FUNCTION_BLOCK FB_MotionAxisNC IMPLEMENTS I_MotionAxis
VAR_INPUT
END_VAR
VAR_OUTPUT
END_VAR
VAR
    {attribute 'no_copy'}
    AxisRef : REFERENCE TO AXIS_REF;
    iMotionAxisCommon : I_MotionAxisCommon;
    iPersistentDataStorage : I_PersistentDataStorage;
    iMotionLogger : I_MotionLogger;

    stAxisParameterSetExposed : ST_AxisParameterSetExposed;

    // This prevent unexpected logical 1 on stMotionStage.bExecute
    nErrorId			: UDINT:=0;
    bHomingBusy			: BOOL;
    bHomingDone			: BOOL;
    fHomePosition : LREAL :=0.0;
    bError				: BOOL;
    sErrorMessage		: STRING;

    fSetPosition	: LREAL;
    fSetVelocity	: LREAL;
    fSetAcceleration	: LREAL := 0.0;
    fSetDeceleration	: LREAL := 0.0;
    fSetJerk	: LREAL := 0.0;
    nHomingMode:ENUM_EpicsHomeCmd :=ENUM_EpicsHomeCmd.NONE;
    eBufferMode	: MC_BufferMode := .MC_BufferMode.MC_Aborting;
    eMoveMode : E_MoveMode;
    sName : STRING;
    // Piezo Motion Control
    tholtime		: TIME := T#10S;
    bBusy : BOOL;
    bDone: BOOL;
    bPowerEnable : BOOL;
    bPowerEnableNegative : BOOL;
    bPowerEnablePositive : BOOL;
    bPowerIsEnabled : BOOL;
    fPowerOverride : LREAL;
    bResetDone : BOOL;
    bHaltDone : BOOL;
    bHomeDone  : BOOL;

    {attribute 'hide'}
    eAxisState : MC_AxisStates;
    // intermediary motion signal: from EPICS interface
    bCmdMoveAbsolute	: BOOL;
    bCmdReset 			: BOOL;
    bCmdHalt 			: BOOL;
    bCmdMoveHome			: BOOL;
    nCommand 		: UINT;
    nCommandData		: UINT;
    nEncoderCount	: UDINT;
    fMoveAbsoluteTargetPosition : LREAL;
    fMoveAbsoluteTargetVelocity : LREAL;
    fMoveAbsoluteTargetAcceleration : LREAL;
    fMoveAbsoluteTargetDeceleration : LREAL;
    fMoveAbsoluteTargetJerk : LREAL;
    fMeasuredAcceleration : LREAL;
    fMeasuredVelocity : LREAL;
    fMeasuredPosition : LREAL;
    fMeasuredPositionDiff : LREAL;

    rtDone 				: R_TRIG;
    rtError				: R_TRIG;
    rtReset				: R_TRIG;
    rtHomed				: R_TRIG;
    ftServo				: F_TRIG;
END_VAR

// Propagate user command to common worker
// 1- Power status
iMotionAxisCOmmon.BufferMode := THIS^.eBufferMode;
iMotionAxisCommon.PowerEnable := THIS^.bPowerEnable;
iMotionAxisCommon.PowerEnableNegative := THIS^.bPowerEnableNegative;
iMotionAxisCommon.PowerEnablePositive := THIS^.bPowerEnablePositive;
iMotionAxisCommon.PowerOverride := THIS^.fPowerOverride;
// 2- Motion commands
iMotionAxisCommon.CommandedHalt := THIS^.bCmdHalt;
iMotionAxisCommon.CommandedReset := THIS^.bCmdReset;
iMotionAxisCommon.CommandedMoveAbsolute := THIS^.bCmdMoveAbsolute;
iMotionAxisCommon.MoveAbsoluteTargetPosition := THIS^.fMoveAbsoluteTargetPosition;
iMotionAxisCommon.MoveAbsoluteTargetVelocity := THIS^.fMoveAbsoluteTargetVelocity;
iMotionAxisCommon.MoveAbsoluteTargetAcceleration := THIS^.fMoveAbsoluteTargetAcceleration;
iMotionAxisCommon.MoveAbsoluteTargetDeceleration := THIS^.fMoveAbsoluteTargetDeceleration;
iMotionAxisCommon.MoveAbsoluteTargetJerk := THIS^.fMoveAbsoluteTargetJerk;

// readbacks and status update from common worker
THIS^.fMeasuredAcceleration := iMotionAxisCommon.MeasuredAcceleration;
THIS^.fMeasuredVelocity := iMotionAxisCommon.MeasuredVelocity;
THIS^.fMeasuredPosition := iMotionAxisCommon.MeasuredPosition;
THIS^.fMeasuredPositionDiff := iMotionAxisCommon.MeasuredPositionDiff;
THIS^.bHaltDone := iMotionAxisCommon.HaltDone;
THIS^.bResetDone := iMotionAxisCommon.ResetDone;
THIS^.bDone := iMotionAxisCommon.MoveAbsoluteDone OR THIS^.HomeDone;
THIS^.bBusy := iMotionAxisCommon.MoveAbsoluteBusy OR THIS^.HomingBusy;
THIS^.bError := iMotionAxisCommon.Error;
THIS^.nErrorId := iMotionAxisCommon.ErrorID;
THIS^.sErrorMessage := iMotionAxisCommon.ErrorMessage;
THIS^.eAxisState := iMotionAxisCommon.AxisState;

// reset cmds if done, error or reset
rtDone(CLK:=bDone);
rtError(CLK:=bError);
rtReset(CLK:=bCmdReset);
IF rtDone.Q OR rtError.Q OR rtReset.Q THEN
    bCmdMoveAbsolute	:= FALSE;
    bCmdReset	:= FALSE;
    bCmdHalt 	:= FALSE;
    bCmdMoveHome	:= FALSE;
END_IF

PROPERTY AxisParameterSetExposed : ST_AxisParameterSetExposed
GET
AxisParameterSetExposed := stAxisParameterSetExposed;
END_GET
END_PROPERTY

PROPERTY AxisState : MC_AxisStates
GET
AxisState := eAxisState;
END_GET
END_PROPERTY

{warning 'Add property implementation'}
PROPERTY BufferMode : MC_BufferMode
SET
BufferMode := eBufferMode;
END_SET
END_PROPERTY

PROPERTY Busy : BOOL
GET
Busy := bBusy;
END_GET
END_PROPERTY

PROPERTY CmdHalt : BOOL
GET
CmdHalt := bCmdHalt;
END_GET
SET
bCmdHalt := CmdHalt;
END_SET
END_PROPERTY

PROPERTY CmdMoveAbsolute : BOOL
GET
CmdMoveAbsolute := bCmdMoveAbsolute;
END_GET
SET
bCmdMoveAbsolute := CmdMoveAbsolute;
END_SET
END_PROPERTY

PROPERTY CmdMoveHome : BOOL
GET
CmdMoveHome := bCmdMoveHome;
END_GET
SET
bCmdMoveHome := CmdMoveHome;
END_SET
END_PROPERTY


PROPERTY CmdReset : BOOL
GET
CmdReset := bCmdReset;
END_GET
SET
bCmdReset := CmdReset;
END_SET
END_PROPERTY

PROPERTY Command : UINT
SET
END_SET
END_PROPERTY

PROPERTY CommandData : UINT
SET
nCommandData := CommandData;
END_SET
END_PROPERTY

PROPERTY Done : BOOL
GET
Done := bDone;
END_GET
END_PROPERTY

PROPERTY EncoderCount : UDINT
GET
EncoderCount := nEncoderCount;
END_GET
END_PROPERTY

PROPERTY Error : BOOL
GET
Error := bError;
END_GET
END_PROPERTY

{warning 'Add property implementation'}
PROPERTY ErrorID : UDINT
GET
ErrorID := nErrorID;
END_GET
END_PROPERTY

{warning 'Add property implementation'}
PROPERTY ErrorMessage : STRING
GET
ErrorMessage := sErrorMessage;
END_GET
END_PROPERTY

//FB_Init is always available implicitly and it is used primarily for initialization.
//The return value is not evaluated. For a specific influence, you can also declare the
//methods explicitly and provide additional code there with the standard initialization
//code. You can evaluate the return value.
METHOD FB_Init: BOOL
VAR_INPUT
    bInitRetains: BOOL; // TRUE: the retain variables are initialized (reset warm / reset cold)
    bInCopyCode: BOOL;  // TRUE: the instance will be copied to the copy code afterward (online change)

    AxisRef : REFERENCE TO AXIS_REF;
    iMotionAxisCommon : I_MotionAxisCommon;
    iPersistentDataStorage : I_PersistentDataStorage;
    iMotionLogger : I_MotionLogger;
END_VAR
THIS^.AxisRef REF= AxisRef;
THIS^.iMotionAxisCommon := iMotionAxisCommon;
THIS^.iPersistentDataStorage := iPersistentDataStorage;
THIS^.iMotionLogger := iMotionLogger;
END_METHOD

PROPERTY HaltDone : BOOL
GET
HaltDone := bHaltDone;
END_GET
END_PROPERTY

{warning 'Add property implementation'}
PROPERTY HomeDone : BOOL
GET
END_GET
END_PROPERTY

{warning 'Add property implementation'}
PROPERTY HomeMode : E_EpicsHomeCmd
GET
END_GET
SET
END_SET
END_PROPERTY

{warning 'Add property implementation'}
PROPERTY HomePosition : LREAL
GET
END_GET
SET
END_SET
END_PROPERTY

{warning 'Add property implementation'}
PROPERTY HomingBusy : BOOL
GET
END_GET
SET
END_SET
END_PROPERTY

{warning 'Add method implementation '}
METHOD InterruptMove
END_METHOD

PROPERTY MeasuredAcceleration : LREAL
GET
MeasuredAcceleration := fMeasuredAcceleration;
END_GET
END_PROPERTY

{warning 'Add property implementation'}
PROPERTY MeasuredPosition : LREAL
GET
MeasuredPosition := fMeasuredPosition;
END_GET
END_PROPERTY

{warning 'Add property implementation'}
PROPERTY MeasuredPositionDiff : LREAL
GET
MeasuredPositionDiff := fMeasuredPositionDiff;
END_GET
END_PROPERTY

PROPERTY MeasuredVelocity : LREAL
GET
MeasuredVelocity := fMeasuredVelocity;
END_GET
END_PROPERTY

{warning 'Add property implementation'}
PROPERTY ModeOfOperation : SINT
GET
END_GET
SET
END_SET
END_PROPERTY

PROPERTY MoveAbsoluteTargetAcceleration : LREAL
GET
MoveAbsoluteTargetAcceleration := fMoveAbsoluteTargetAcceleration;
END_GET
SET
fMoveAbsoluteTargetAcceleration := MoveAbsoluteTargetAcceleration;
END_SET
END_PROPERTY

PROPERTY MoveAbsoluteTargetDeceleration : LREAL
GET
MoveAbsoluteTargetDeceleration := fMoveAbsoluteTargetDeceleration;
END_GET
SET
fMoveAbsoluteTargetDeceleration := MoveAbsoluteTargetDeceleration;
END_SET
END_PROPERTY

PROPERTY MoveAbsoluteTargetJerk : LREAL
GET
MoveAbsoluteTargetJerk := fMoveAbsoluteTargetJerk;
END_GET
SET
fMoveAbsoluteTargetJerk := MoveAbsoluteTargetJerk;
END_SET
END_PROPERTY

PROPERTY MoveAbsoluteTargetPosition : LREAL
GET
MoveAbsoluteTargetPosition := fMoveAbsoluteTargetPosition;
END_GET
SET
fMoveAbsoluteTargetPosition := MoveAbsoluteTargetPosition;
END_SET
END_PROPERTY

PROPERTY MoveAbsoluteTargetVelocity : LREAL
GET
MoveAbsoluteTargetVelocity := fMoveAbsoluteTargetVelocity;
END_GET
SET
fMoveAbsoluteTargetVelocity := MoveAbsoluteTargetVelocity;
END_SET
END_PROPERTY

PROPERTY MoveMode : E_MoveMode
GET
MoveMode := eMoveMode;
END_GET
SET
eMoveMode := MoveMode;
END_SET
END_PROPERTY

PROPERTY Name : STRING
GET
Name := sName;
END_GET
SET
sName := Name;
END_SET
END_PROPERTY

{warning 'Add property implementation'}
PROPERTY NegativeMotionIsEnabled : BOOL
GET
END_GET
END_PROPERTY

{warning 'Add property implementation'}
PROPERTY PositiveMotionIsEnabled : BOOL
GET
END_GET
END_PROPERTY

PROPERTY PowerEnable : BOOL
GET
PowerEnable := bPowerEnable;
END_GET
SET
bPowerEnable := PowerEnable;
END_SET
END_PROPERTY

PROPERTY PowerEnableNegative : BOOL
GET
PowerEnableNegative := bPowerEnableNegative;
END_GET
SET
bPowerEnableNegative := PowerEnableNegative;
END_SET
END_PROPERTY

PROPERTY PowerEnablePositive : BOOL
GET
PowerEnablePositive := bPowerEnablePositive;
END_GET
SET
bPowerEnablePositive := PowerEnablePositive;
END_SET
END_PROPERTY

{warning 'Add property implementation'}
PROPERTY PowerIsEnabled : BOOL
GET
PowerIsEnabled := bPowerIsEnabled;
END_GET
END_PROPERTY

{warning 'Add property implementation'}
PROPERTY PowerOverride : LREAL
GET
PowerOverride := fPowerOverride;
END_GET
SET
fPowerOverride := PowerOverride;
END_SET
END_PROPERTY

PROPERTY ResetDone : BOOL
GET
ResetDone := bResetDone ;
END_GET
END_PROPERTY

{warning 'Add property implementation'}
PROPERTY Servo : BOOL
GET
END_GET
SET
END_SET
END_PROPERTY

(*
    Check all post condition before updating bCommandedMoveAbsolute
    The implmentatation will depend on the axis type
    DS402 NC/Direct axis : Implementation need to check that the drive is in the correct mode before initaiting the move then set bCommandedMoveAbsolute
    MP NC axis : will immediately write to bCommandedMoveAbsolute
*)
METHOD StartMove : BOOL
VAR_INPUT
END_VAR
CASE eMoveMode OF
    E_MoveMode.DISCRETE:
        iMotionAxisCommon.CommandedMoveAbsolute := THIS^.bCmdMoveAbsolute;
    E_MoveMode.HOMING:
    THIS^.bCmdMoveHome := TRUE;
END_CASE

// for typical NC axis no further test is needed
StartMove := TRUE;
END_METHOD

{warning 'Add method implementation '}
METHOD StopMove
END_METHOD

END_FUNCTION_BLOCK

(* stored: Version 1.1.0.1
   POU FB_MotionAxisNC: Id {abd0b982-5130-4244-8207-eba0b3246906}, SpecialFunc None
   Property AxisParameterSetExposed: Id {384b2d0e-5f4f-4936-8350-ceae816b150e}
   Get Get: Id {c87f54a1-a5eb-49de-8441-7a2ad0ec72de}
   Property AxisState: Id {904290e4-8519-49b9-badc-b3e1713daec6}
   Get Get: Id {ccec9d39-634d-4098-ae3d-57765a8e4217}
   Property BufferMode: Id {2c65028d-a104-4e19-872f-4dd701e61531}
   Set Set: Id {6e4cbde5-d3db-4fb0-90d0-8e798f99604b}
   Property Busy: Id {8b5e8894-c876-41b1-9e2c-980090299d06}
   Get Get: Id {0589f453-0019-4df2-87e7-619c947d4d89}
   Property CmdHalt: Id {18dd0b55-37ec-4bc8-a0d2-55b6db6a152f}
   Get Get: Id {a8673054-4564-489f-91d8-dc779daec553}
   Set Set: Id {bb6fa02c-7a76-469a-ae3d-d5fddedf6fd7}
   Property CmdMoveAbsolute: Id {8ba6543e-9bbe-4c2c-985e-e7797189c137}
   Get Get: Id {10aedfd5-412b-492b-b988-266d9f40addf}
   Set Set: Id {1edbd315-9001-4619-ac2e-1d29105a5138}
   Property CmdMoveHome: Id {9dc329c6-3e63-4e47-98ec-522d097b78c3}
   Get Get: Id {497b21ae-b468-49fa-a678-10ae542a591a}
   Set Set: Id {d15709fd-f925-450c-9e97-7665b59292b5}
   Property CmdReset: Id {70bf962c-f201-42b0-acce-f42a534f0e53}
   Get Get: Id {400e310e-bcfd-485d-b2ea-e2b29fff54cb}
   Set Set: Id {d260d983-2678-4bcb-9070-7db5839a6fca}
   Property Command: Id {1bfbf561-216d-484d-b0f5-59e0d5d323f0}
   Set Set: Id {7b937c3c-33f5-4681-a1fc-8827e5918112}
   Property CommandData: Id {2f61ec8e-7923-460c-bb0d-1c4f6bf683f9}
   Set Set: Id {7ac59737-5819-446b-adb3-fad8bc24c252}
   Property Done: Id {7dfea87f-91d0-4696-931e-3f0a58f16ac5}
   Get Get: Id {b56b7cc9-86b2-4c3c-bc8f-26dc7bf2e509}
   Property EncoderCount: Id {cd5917d9-7633-485a-80ea-f12e3b700502}
   Get Get: Id {929c4496-fbe3-4004-b896-c4d0a35e2293}
   Property Error: Id {4da1c0dd-304a-4f96-9c35-e21861c7cc5a}
   Get Get: Id {cb4df7cd-44c4-45b9-9d32-a492dc206cc9}
   Property ErrorID: Id {a9cd6d81-3a12-4ea6-a064-5e3b63b03982}
   Get Get: Id {5ddc443f-6d54-4a83-a527-83e86fdb72b0}
   Property ErrorMessage: Id {aeeaa0d1-15f3-4400-b508-44a15c83d1d3}
   Get Get: Id {5f52a084-10af-4e78-8941-03dd3f8cdb45}
   Method FB_Init: Id {0f22422e-d0d7-4f19-ba6a-909d8434ca89}
   Property HaltDone: Id {3e07c920-60e0-4810-a3dc-4b8f36ba148b}
   Get Get: Id {fbe1db8b-e303-42af-aa5c-f6f6b3b3c9b9}
   Property HomeDone: Id {58d55820-86b5-4ff6-b9aa-fa09a9de7d99}
   Get Get: Id {260eedc9-efbe-40a9-af5a-fbf7edde8655}
   Property HomeMode: Id {66c6b98c-e856-4ec1-8f29-50ec1e680ce0}
   Get Get: Id {0682ce34-446a-4ad8-b130-0e89580447ca}
   Set Set: Id {b74d39df-3a6a-4831-ba53-397fffaa80dd}
   Property HomePosition: Id {d1dcd6fe-6238-4a59-bf71-904087434b65}
   Get Get: Id {4e265816-2c35-4ac5-8efe-9b820a4659d3}
   Set Set: Id {a862b520-5642-43f4-a7dd-d8bbc5e09cf7}
   Property HomingBusy: Id {a424505c-197f-4965-8907-a5bb521bca80}
   Get Get: Id {a11f36be-6698-4aa3-bdba-8e3d5f05b66b}
   Set Set: Id {53b6540f-6a73-446f-bbcb-8f8c3abb9b70}
   Method InterruptMove: Id {f2042942-3668-4c52-a5a8-4eafd072cc2d}
   Property MeasuredAcceleration: Id {7e81f087-a061-41fe-adda-cdd75fb8d3b7}
   Get Get: Id {1fb1b26a-c93f-4978-8c85-5aca7ba005c8}
   Property MeasuredPosition: Id {06e7e9c6-bd4c-49c7-b334-4675cee48bbf}
   Get Get: Id {ca4f3174-19ae-4b41-a8aa-372784a3ac03}
   Property MeasuredPositionDiff: Id {86588116-492b-4d24-b0c9-5d4dc4e8e3ad}
   Get Get: Id {ae3b9f00-5a1d-497e-9d73-65845bc824fa}
   Property MeasuredVelocity: Id {df9982a2-284d-4e07-a730-805522796a88}
   Get Get: Id {3ce526bf-887f-4f07-b397-c7b40bc7ea9d}
   Property ModeOfOperation: Id {d6016f57-7749-495f-9da1-2128cd309525}
   Get Get: Id {5e91de21-580c-4d8c-ae79-241c60a96b06}
   Set Set: Id {440ba54b-0f2f-450f-93d8-7075809b65a2}
   Property MoveAbsoluteTargetAcceleration: Id {b48e2972-c8fc-4dcb-98ca-4d1a8db067eb}
   Get Get: Id {b4223350-cd20-4630-afad-34e2dbadc01d}
   Set Set: Id {54fac66c-8ef0-4ab6-bdb4-718acd17e847}
   Property MoveAbsoluteTargetDeceleration: Id {7b23395a-f43a-485c-b091-6dede893ab02}
   Get Get: Id {f24320ab-f202-4085-84c1-f054b91161dc}
   Set Set: Id {d6625075-b652-49cc-98f2-02d8ddf9344d}
   Property MoveAbsoluteTargetJerk: Id {c43e9e4f-a17b-498d-b040-dae732b65331}
   Get Get: Id {1eeace55-74bc-4ea1-94df-7108761c4113}
   Set Set: Id {f3a9efcc-941a-4b43-a0e4-107ff48cc40d}
   Property MoveAbsoluteTargetPosition: Id {2e86d8a8-f29b-43d2-9bdb-96af59865924}
   Get Get: Id {995d8422-2ec1-4c5a-a91a-37f299f60908}
   Set Set: Id {976ecf4d-3776-46dd-a3e3-a68132688cc5}
   Property MoveAbsoluteTargetVelocity: Id {e615d560-a621-4c43-b5ac-5ce3d0036d44}
   Get Get: Id {4a4935af-81be-4856-8f74-33e494892137}
   Set Set: Id {c4f65d76-2089-4b5a-803f-74876d126f9e}
   Property MoveMode: Id {2349362a-d96e-441f-980a-966606218489}
   Get Get: Id {53f09a95-d6df-464c-9a62-eb6e0e8899e9}
   Set Set: Id {a48dfab9-73bb-4b00-ab53-c30621597c3d}
   Property Name: Id {17cf3a61-c148-4cf5-b5a3-52380a5358bf}
   Get Get: Id {481d2186-b92d-4a40-b4d4-c39ddfa9d67b}
   Set Set: Id {e85db46e-2038-4454-b89c-e98feb9fb5a3}
   Property NegativeMotionIsEnabled: Id {6a32db5d-750b-4ff0-b32d-784834aacf25}
   Get Get: Id {4f3f9292-d844-4954-8bfd-d20b0081868f}
   Property PositiveMotionIsEnabled: Id {0ebc8e3d-fb03-417b-abdf-abbfb62dbc04}
   Get Get: Id {cc5c0f81-da44-45e3-9e8f-7302b534ba4a}
   Property PowerEnable: Id {e52fdcf1-093e-480d-8441-6cf95fbaa158}
   Get Get: Id {9018b8fd-888e-4852-a2a5-77f407619e51}
   Set Set: Id {3a420c38-e9e8-4911-ab2a-175fac23918e}
   Property PowerEnableNegative: Id {00926e8e-1515-4c4c-9953-c30e7aebbb2c}
   Get Get: Id {7c705b7b-c9c8-4748-b171-c39863a607ce}
   Set Set: Id {d65cba3d-5353-412c-aa27-f290efc4beae}
   Property PowerEnablePositive: Id {891bfa66-c294-4d3d-9609-6d5161e8cb67}
   Get Get: Id {1646fbff-f59b-4bf1-9cb1-5a3c106477cf}
   Set Set: Id {4b90045e-6809-4ffb-8548-9ae5478fd00c}
   Property PowerIsEnabled: Id {a4686680-607b-4188-9777-0f0c86ac0492}
   Get Get: Id {4a5c4c22-1a41-41a6-8532-cad8d18168b9}
   Property PowerOverride: Id {4fee9dae-6fa1-4dd8-96d5-908a0d05341d}
   Get Get: Id {a3952dac-e1e7-4fdb-a522-10de1ed7f294}
   Set Set: Id {0efa8f22-e731-48e2-924b-58b213053e9f}
   Property ResetDone: Id {4627e064-5c4d-4edb-9e16-cbe14d9d786e}
   Get Get: Id {1cb04972-43f8-42e9-b15b-7a40ec5b6358}
   Property Servo: Id {f22af3bc-c2ef-4742-95ad-ccee48f4f0fc}
   Get Get: Id {2a5500de-6503-4ee9-ac20-949ef8f86761}
   Set Set: Id {085ee16c-1c78-49fb-8996-52d5b83452a0}
   Method StartMove: Id {ddca3259-b438-4587-9e7c-acef815aa982}
   Method StopMove: Id {df32edec-47df-4332-b762-89a58ea420b3} *)
